FUNCTION_BLOCK Hutschienenmoped_XL_8_AI (* Service Interface Function Block Type *)
  (* Function: All Inputs; Description: this maps to ID *)
  (* Version 1.0, 2018-12-05, Jose Cabral *)
  (* Version 1.1, 2022-08-04, Franz Höpfinger, HR Agrartechnik GmbH *)
  (* Version 1.2, 2023-01-05, Franz Höpfinger, HR Agrartechnik GmbH *)
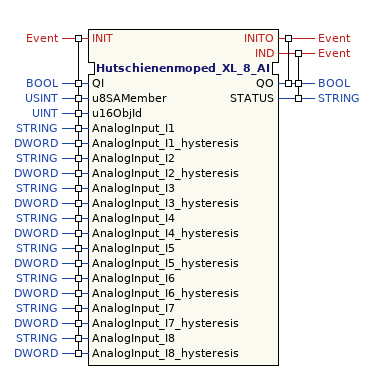
  EVENT_INPUT
    INIT WITH QI, u8SAMember, u16ObjId, AnalogInput_I1, AnalogInput_I1_hysteresis, AnalogInput_I2, AnalogInput_I2_hysteresis, AnalogInput_I3, AnalogInput_I3_hysteresis, AnalogInput_I4, AnalogInput_I4_hysteresis, AnalogInput_I5, AnalogInput_I5_hysteresis, AnalogInput_I6, AnalogInput_I6_hysteresis, AnalogInput_I7, AnalogInput_I7_hysteresis, AnalogInput_I8, AnalogInput_I8_hysteresis; (* Service Initialization *)
  END_EVENT
  EVENT_OUTPUT
    INITO WITH QO; (* Initialization Confirm *)
    IND WITH QO, STATUS; (* Indication from Resource *)
  END_EVENT
  VAR_INPUT
    QI : BOOL; (* Event Input Qualifier *)
    u8SAMember : USINT := GLOBAL; (* Dummy !, set to GLOBAL if in doubt. OFF deactivates FB. *)
    u16ObjId : UINT := ID_NULL; (* Dummy ! set to ID_NULL if in Doubt. ID_OFF deactivates FB. *)
    AnalogInput_I1 : STRING; (* Identifier for Input 1 *)
    AnalogInput_I1_hysteresis : DWORD;
    AnalogInput_I2 : STRING; (* Identifier for Input 2 *)
    AnalogInput_I2_hysteresis : DWORD;
    AnalogInput_I3 : STRING; (* Identifier for Input 3 *)
    AnalogInput_I3_hysteresis : DWORD;
    AnalogInput_I4 : STRING; (* Identifier for Input 4 *)
    AnalogInput_I4_hysteresis : DWORD;
    AnalogInput_I5 : STRING; (* Identifier for Input 5 *)
    AnalogInput_I5_hysteresis : DWORD;
    AnalogInput_I6 : STRING; (* Identifier for Input 6 *)
    AnalogInput_I6_hysteresis : DWORD;
    AnalogInput_I7 : STRING; (* Identifier for Input 7 *)
    AnalogInput_I7_hysteresis : DWORD;
    AnalogInput_I8 : STRING; (* Identifier for Input 8 *)
    AnalogInput_I8_hysteresis : DWORD;
  END_VAR
  VAR_OUTPUT
    QO : BOOL; (* Event Output Qualifier *)
    STATUS : STRING; (* Service Status *)
  END_VAR
END_FUNCTION_BLOCK
